(* IEC 61131-3 sources: ecmccfg/examples/PSI/lab_setup/stepper_bissc/cfg, 1 file *)

(* ---- test.plc ---- *)
VAR
  myPLC: ${SELF};
  myAxis: ax1;
  mySlave: ${M}.s${S_ID};
END_VAR

if(myPLC.firstscan){
  println('Starting up!!!!');
};

println('position: ', mySlave.positionActual01);
